(*

.. <legal notes>

legal notes
=================
| SPDX-FileCopyrightText: © 2025 Oleksandr Tiutyk <trofimich@gmail.com>
| SPDX-License-Identifier: LGPL-3.0-only
| For details check: LGPL-3.0-only_

.. _LGPL-3.0-only: https://www.gnu.org/licenses/lgpl-3.0.en.html

.. </legal notes>

*)

{attribute 'no_explicit_call' := 'do not call this function block directly'} 
{attribute 'enable_dynamic_creation'}
FUNCTION_BLOCK IfElseActivity EXTENDS Activity IMPLEMENTS IIfElseActivity
VAR
	{attribute 'OPC.UA.DA' := '0'}
	_ClassName : STRING := __POUNAME();

	{attribute 'OPC.UA.DA' := '0'}
	_Condition : ICondition;	

	{attribute 'OPC.UA.DA' := '0'}
	_TrueActivity : IActivity;
	
	{attribute 'OPC.UA.DA' := '0'}
	_FalseActivity : IActivity;

	{attribute 'OPC.UA.DA' := '0'}
	_CurrentActivity : IActivity;
END_VAR

{attribute 'monitoring' := 'call'}
PROPERTY ClassName : STRING
GET
ClassName := _ClassName;
END_GET
END_PROPERTY

{attribute 'monitoring' := 'call'}
PROPERTY FINAL Condition : ICondition
GET
Condition := _Condition;
END_GET
SET
_Condition := Condition;
END_SET
END_PROPERTY

METHOD Configure
VAR_INPUT
	condition : ICondition; 
	trueActivity : IActivity;
	falseActivity : IActivity;
END_VAR
VAR
	argumentNullException : Core.ArgumentNullException;
END_VAR
IF condition = 0 THEN
	argumentNullException.Throw(NamespaceName, ClassName, __POUNAME(), __POSITION(), 'condition');
END_IF

_Condition := condition;
_TrueActivity := trueActivity;
_FalseActivity := falseActivity;
END_METHOD

{attribute 'monitoring' := 'call'}
PROPERTY FINAL CurrentActivity : IActivity
GET
CurrentActivity := _CurrentActivity;
END_GET
END_PROPERTY

{attribute 'monitoring' := 'call'}
PROPERTY FINAL FalseActivity : IActivity
GET
FalseActivity := _FalseActivity;
END_GET
SET
_FalseActivity := FalseActivity;
END_SET
END_PROPERTY

{attribute 'monitoring' := 'call'}
PROPERTY NamespaceName : STRING
GET
NamespaceName := CurrentNamespace.Name;
END_GET
END_PROPERTY

METHOD PROTECTED OnAborting 
VAR_INPUT
	isStart : BOOL;
END_VAR
VAR_OUTPUT
	done : BOOL;
END_VAR
VAR
	conditionIsNullException : Core.NullReferenceException;
END_VAR
IF _Condition = 0 THEN
	conditionIsNullException.Throw(NamespaceName, ClassName, __POUNAME(), __POSITION(), 'Condition');
END_IF

IF _CurrentActivity = 0 OR_ELSE NOT _CurrentActivity.Busy THEN
	done := TRUE;
	RETURN;
END_IF

IF isStart THEN
	_CurrentActivity.StartAbort();
ELSE
	_CurrentActivity.Execute();
END_IF
	
done := NOT _CurrentActivity.Busy;
END_METHOD

METHOD PROTECTED OnRunning 
VAR_INPUT
	isStart : BOOL;
END_VAR
VAR_OUTPUT
	done : BOOL;
END_VAR
VAR
	workflowVariable : Core.GENERIC_VALUE;
	
	conditionIsNullException : Core.NullReferenceException;
END_VAR
IF _Condition = 0 THEN
	conditionIsNullException.Throw(NamespaceName, ClassName, __POUNAME(), __POSITION(), 'Condition');
END_IF

IF isStart THEN
	IF _Condition.Evaluate(THIS^) THEN
		_CurrentActivity := _TrueActivity;
	ELSE
		_CurrentActivity := _FalseActivity;
	END_IF
END_IF

IF _CurrentActivity <> 0 THEN
	IF isStart THEN
		_CurrentActivity.Start();
	ELSE
		_CurrentActivity.Execute();
	END_IF
	
	done := NOT _CurrentActivity.Busy;
ELSE
	done := TRUE;
END_IF
END_METHOD

{attribute 'monitoring' := 'call'}
PROPERTY Size : ULINT
GET
Size := XSIZEOF(THIS^);
END_GET
END_PROPERTY

{attribute 'monitoring' := 'call'}
PROPERTY FINAL TrueActivity : IActivity
GET
TrueActivity := _TrueActivity;
END_GET
SET
_TrueActivity := TrueActivity;
END_SET
END_PROPERTY

END_FUNCTION_BLOCK

(* stored: Version 1.1.0.1
   POU IfElseActivity: Id {da8ca86c-872c-4aea-b306-b93e7546e465}, SpecialFunc None
   Folder Overriden: Id {2eaaea99-11a7-47d3-bce1-f5e4002d484d}
   Property ClassName: Id {52ba2f22-b051-4c36-b8e4-569e32a5fbcd}
   Get Get: Id {8f1e88e3-d595-4f40-b825-4fa1aa0576b5}
   Property Condition: Id {d6d3b9ec-abfb-47ac-b244-779a1768e5d1}
   Get Get: Id {df58c0b6-ab5e-42d6-b2fa-3e5cf61a4d91}
   Set Set: Id {f33f3eb2-9a27-4ee9-818e-527084aede90}
   Method Configure: Id {c77bc6c7-c58c-40d4-b1de-9802d060e7cc}
   Property CurrentActivity: Id {bb159f09-2ec7-4d87-8336-5235c12ce96e}
   Get Get: Id {bdfbe9b8-d360-4588-aec6-083acd66706e}
   Property FalseActivity: Id {df0b0194-8599-4654-a290-f9364f04d58a}
   Get Get: Id {629e68a7-86ee-4b70-8f7f-2a06679d8b24}
   Set Set: Id {c40d09b3-f46c-4a41-bd1a-37eac419410d}
   Property NamespaceName: Id {bdec18b4-d519-428c-889d-15c7cbdf3042}
   Get Get: Id {ab9a48f4-7b32-4f0f-8716-2ee04a15c52b}
   Method OnAborting: Id {b44a164a-4eac-46c0-b278-02b556ce0ce5}
   Method OnRunning: Id {176adfb9-e622-4478-9575-8d7951a3282b}
   Property Size: Id {65b8bb80-4ccf-4179-b71f-fb77944444bc}
   Get Get: Id {144dcbe8-489f-4b59-99a0-a091c9248ba0}
   Property TrueActivity: Id {df748dd9-c1bb-4689-8969-3592e599e9f6}
   Get Get: Id {ddad71d3-ec7a-4afd-9f95-fbeb07e458e3}
   Set Set: Id {70915f8a-c0f8-40ef-b852-7d88bd336ae7} *)
